FUNCTION_BLOCK fb_undock
VAR_INPUT
END_VAR
VAR_OUTPUT
END_VAR
VAR
	step: INT;
	unLock: fb_toggleVal;
END_VAR

CASE step OF
	0:
		IF NOT tcin.ProxUp THEN
			unLock(IN:= TRUE);
			unLock.IN := FALSE;
			cntrlstate.piston_moving := TRUE;
			step := 1;
		END_IF
	1: 
		IF tcin.ProxUp AND tcin.ProxUp THEN
			 cntrlstate.undock := TRUE;
			 cntrlstate.piston_moving := FALSE;
			 step := 0;
		END_IF
	99:
		//ERROR HANDLING
END_CASE
unLock();
(*
CASE step OF
	0:
		IF tcin.ProxDwn THEN
			unLock(IN:= TRUE);
			unLock.IN := FALSE;
			cntrlstate.piston_moving := TRUE;
			step := 1;
		END_IF
	1: 
		IF tcin.ProxUp AND NOT tcin.ProxDwn THEN
			 cntrlstate.undock := TRUE;
			 cntrlstate.piston_moving := FALSE;
			 step := 0;
		END_IF
	99:
		//ERROR HANDLING
END_CASE
unLock();*)

END_FUNCTION_BLOCK

(* stored: Version 1.1.0.1, ProductVersion 3.1.4024.5
   POU fb_undock: Id {fe6299cd-40da-4124-8f05-58cfe31f1879}, SpecialFunc None *)
